INTERFACE IF_DriveVariableVel

PROPERTY bBOTTOM : BOOL
GET
END_GET
END_PROPERTY

PROPERTY bTOP : BOOL
GET
END_GET
END_PROPERTY

METHOD lifEnable
VAR_INPUT
END_VAR
END_METHOD

METHOD liftDisable
VAR_INPUT
END_VAR
END_METHOD

METHOD moveVarSpeed
VAR_INPUT
	nSetVelocity : INT;
	eDirection : LiftMovingDirection;
END_VAR
END_METHOD

METHOD stop
VAR_INPUT
END_VAR
END_METHOD

END_INTERFACE

(* stored: Version 1.1.0.1, ProductVersion 3.1.4024.6
   Itf IF_DriveVariableVel: Id {f26f961d-e895-426c-987f-bb7572460cb9}
   Property bBOTTOM: Id {77cb1934-0184-4720-b6b9-4ec73f8015e7}
   Get Get: Id {c5596dfa-854f-4c11-938f-c3b4dec469ef}
   Property bTOP: Id {44738e9d-27ff-4c4c-be13-b184ac41aa3b}
   Get Get: Id {a28a6308-baf2-4f55-b4b6-2fcf2efed39d}
   Method lifEnable: Id {579038fa-9827-4a68-a04b-faabe1ad189d}
   Method liftDisable: Id {f77b9e9f-71f5-463a-93a5-9aeb93f830a8}
   Method moveVarSpeed: Id {ebbb665d-2d75-4d85-ac0e-eada4eb83528}
   Method stop: Id {d5b4144c-1790-4954-98b7-1986d51e617b} *)
